// SIMATIC S7-200 project (STEP 7-Micro/WIN), CPU 224XP REL 02.01

SYMBOL_TABLE USUARIO1
P_MARCHA         I0.0
P_PARO           I0.1
P_CAMBIO_DE_GIRO I0.2
TRI_LINEA        Q0.0
TRI_ESTRELLA     Q0.1
TRI_TRIANGULO    Q0.2
CINTA_1          Q0.3
CINTA_2_IZQUIERDAS Q0.4
CINTA_2_DERECHAS Q0.5
END_SYMBOL_TABLE

ORGANIZATION_BLOCK PRINCIPAL:OB1
TITLE=COMENTARIOS DEL PROGRAMA
BEGIN
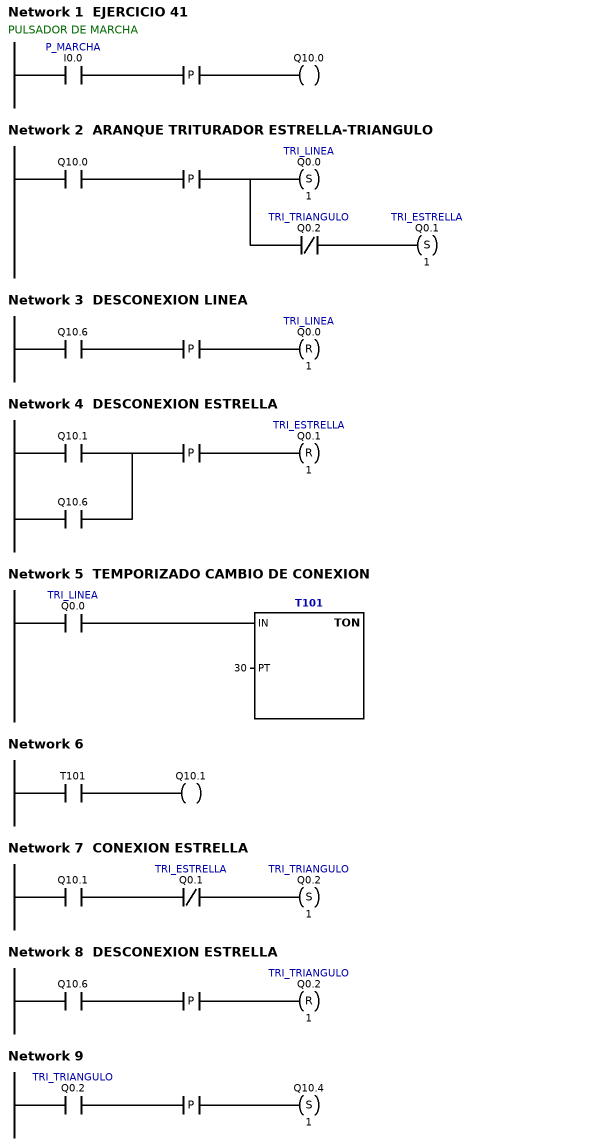
Network 1 // EJERCICIO 41

// PULSADOR DE MARCHA
LD     P_MARCHA:I0.0
EU
=      Q10.0
Network 2 // ARANQUE TRITURADOR ESTRELLA-TRIANGULO
LD     Q10.0
EU
S      TRI_LINEA:Q0.0, 1
AN     TRI_TRIANGULO:Q0.2
S      TRI_ESTRELLA:Q0.1, 1
Network 3 // DESCONEXION LINEA 
// (network saved uncompiled; LAD cells follow)
// row 0: c0 -| |- Q10.6  c1 -|P|-  c2 -(R) TRI_LINEA:Q0.0, 1
Network 4 // DESCONEXION ESTRELLA
// (network saved uncompiled; LAD cells follow)
// row 0: c0 -| |- Q10.1 v  c1 -|P|-  c2 -(R) TRI_ESTRELLA:Q0.1, 1
// row 1: c0 -| |- Q10.6 ^
Network 5 // TEMPORIZADO CAMBIO DE CONEXION
LD     TRI_LINEA:Q0.0
TON    T101, 30
Network 6
// (network saved uncompiled; LAD cells follow)
// row 0: c0 -| |- T101  c1 -( ) Q10.1
Network 7 // CONEXION ESTRELLA
LD     Q10.1
AN     TRI_ESTRELLA:Q0.1
S      TRI_TRIANGULO:Q0.2, 1
Network 8 // DESCONEXION ESTRELLA
LD     Q10.6
EU
R      TRI_TRIANGULO:Q0.2, 1
Network 9
LD     TRI_TRIANGULO:Q0.2
EU
S      Q10.4, 1
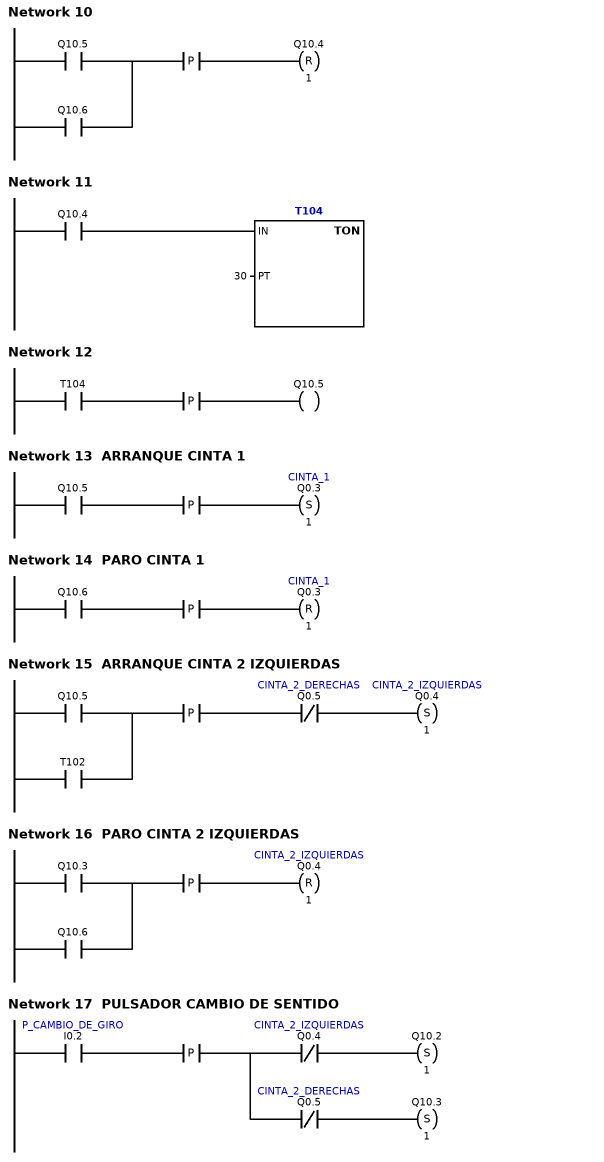
Network 10
LD     Q10.5
O      Q10.6
EU
R      Q10.4, 1
Network 11
LD     Q10.4
TON    T104, 30
Network 12
LD     T104
EU
=      Q10.5
Network 13 // ARRANQUE CINTA 1 
LD     Q10.5
EU
S      CINTA_1:Q0.3, 1
Network 14 // PARO CINTA 1 
LD     Q10.6
EU
R      CINTA_1:Q0.3, 1
Network 15 // ARRANQUE CINTA 2 IZQUIERDAS
// (network saved uncompiled; LAD cells follow)
// row 0: c0 -| |- Q10.5 v  c1 -|P|-  c2 -|/|- CINTA_2_DERECHAS:Q0.5  c3 -(S) CINTA_2_IZQUIERDAS:Q0.4, 1
// row 1: c0 -| |- T102 ^
Network 16 // PARO CINTA 2 IZQUIERDAS
LD     Q10.3
O      Q10.6
EU
R      CINTA_2_IZQUIERDAS:Q0.4, 1
Network 17 // PULSADOR CAMBIO DE SENTIDO
LD     P_CAMBIO_DE_GIRO:I0.2
EU
LPS
AN     CINTA_2_IZQUIERDAS:Q0.4
S      Q10.2, 1
LPP
AN     CINTA_2_DERECHAS:Q0.5
S      Q10.3, 1
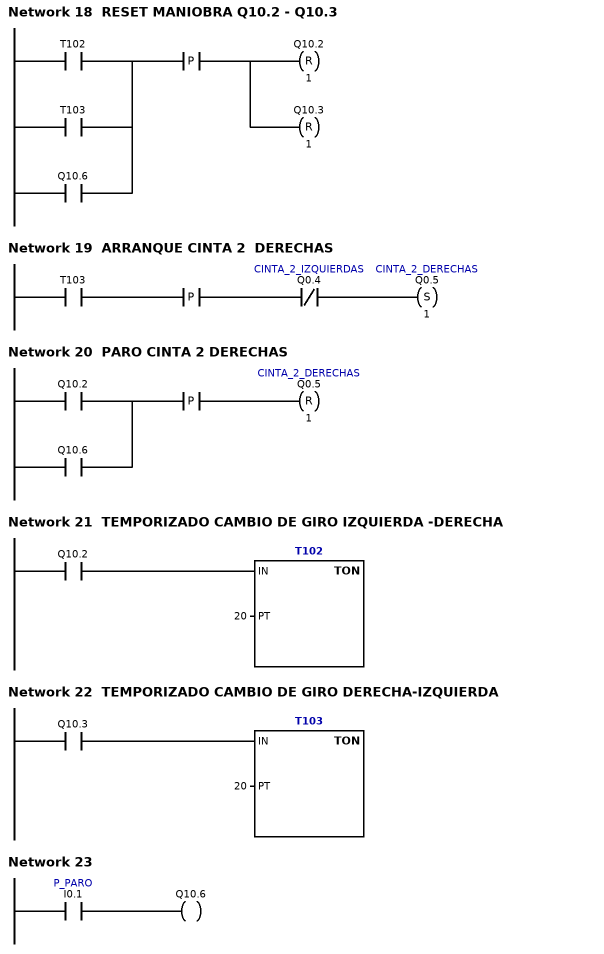
Network 18 // RESET MANIOBRA Q10.2 - Q10.3
LD     T102
O      T103
O      Q10.6
EU
R      Q10.2, 1
R      Q10.3, 1
Network 19 // ARRANQUE CINTA 2  DERECHAS
LD     T103
EU
AN     CINTA_2_IZQUIERDAS:Q0.4
S      CINTA_2_DERECHAS:Q0.5, 1
Network 20 // PARO CINTA 2 DERECHAS
LD     Q10.2
O      Q10.6
EU
R      CINTA_2_DERECHAS:Q0.5, 1
Network 21 // TEMPORIZADO CAMBIO DE GIRO IZQUIERDA -DERECHA
LD     Q10.2
TON    T102, 20
Network 22 // TEMPORIZADO CAMBIO DE GIRO DERECHA-IZQUIERDA
LD     Q10.3
TON    T103, 20
Network 23
LD     P_PARO:I0.1
=      Q10.6
END_ORGANIZATION_BLOCK
